TYPE Clamp :
STRUCT
	Open_Command:BOOL;
	Close_Command:BOOL;
	Opened_Switch_ON:BOOL;
	Closed_Switch_ON:BOOL;
	Jam_Fault:BOOL;
	Air_Pres_OK:BOOL;
	
END_STRUCT
END_TYPE

(* stored: Version 1.1.0.1, ProductVersion 3.1.4024.12
   DUT Clamp: Id {71ad9021-a25e-408f-b4f8-bced98dbac2e} *)
